SUBAPPLICATION F_PWM_PERCENT_TO_RAW (* PWM-Sollwert-Anteil (REAL 0.0-1.0) in Fieldbus-Rohwert (DINT, 0-64255) umrechnen, fuer RampLimitFS.PV *)
  (* Standard: 61499-2 *)
  (* Version 1.0, 2026-08-28, franz *)
  PACKAGE MyLib::sys;
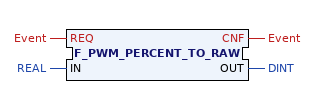
  EVENT_INPUT
    REQ; (* Normal Execution Request *)
  END_EVENT
  EVENT_OUTPUT
    CNF; (* Execution Confirmation *)
  END_EVENT
  VAR_INPUT
    IN : REAL; (* Sollwert-Anteil 0.0-1.0 (nicht Prozent 0-100!), z.B. RampLimitFS-Sollwert / 100.0 *)
  END_VAR
  VAR_OUTPUT
    OUT : DINT; (* Fieldbus-Rohwert 0-64255 (0x0000-0xFAFF, SAE J1939/ISO 11783 VALID_SIGNAL_W), fuer RampLimitFS.PV *)
  END_VAR
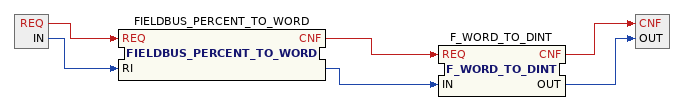
  FBS
    FIELDBUS_PERCENT_TO_WORD : eclipse4diac::signalprocessing::FIELDBUS_PERCENT_TO_WORD;
    F_WORD_TO_DINT : iec61131::conversion::F_WORD_TO_DINT;
  END_FBS
  EVENT_CONNECTIONS
    FIELDBUS_PERCENT_TO_WORD.CNF TO F_WORD_TO_DINT.REQ;
    REQ TO FIELDBUS_PERCENT_TO_WORD.REQ;
    F_WORD_TO_DINT.CNF TO CNF;
  END_CONNECTIONS
  DATA_CONNECTIONS
    FIELDBUS_PERCENT_TO_WORD. TO F_WORD_TO_DINT.IN;
    IN TO FIELDBUS_PERCENT_TO_WORD.RI;
    F_WORD_TO_DINT.OUT TO OUT;
  END_CONNECTIONS
END_SUBAPPLICATION
